TYPE ServicesTimingIOParts :
STRUCT
	///Coupler
	coupler: EtherCatDevice;
	///Slot 1
	slot1: EtherCatDevice;
	///Slot 2
	slot2: EtherCatDevice;
END_STRUCT
END_TYPE

(* stored: Version 1.1.0.1, ProductVersion 3.1.4019.2
   DUT ServicesTimingIOParts: Id {f06a4a54-9a64-4a39-a723-4459559723b6} *)
